Yaskawa INFORM job: X2_DOD_HARDOX_2(90,0).JBI

/JOB
//NAME X2_DOD_HARDOX_2(90,0)
//POS
///NPOS 304,304,304,21,0,0
///TOOL 0
///POSTYPE PULSE
///PULSE
C00000=3322,-122452,-100913,-73,83322,449
C00001=-124273,-75019,-76743,-2114,92937,4431
C00002=-124273,-75019,-76743,-2114,92937,4431
C00003=-142747,-87673,-78422,-11081,73870,-1911
C00004=-145871,-78515,-73342,-10252,75010,-3119
C00005=-145871,-78057,-71113,-10305,73892,-3025
C00006=-145871,-78160,-71592,-10294,74129,-3045
C00007=-146817,-82702,-73614,-10112,72935,-3281
C00008=-146817,-82536,-72956,-10129,72622,-3254
C00009=-146351,-80344,-71991,-10217,73205,-3137
C00010=-146503,-81415,-73793,-10153,73736,-3236
C00011=-173681,-53943,-60859,-2823,77659,-12885
C00012=-172671,-51589,-58765,-3102,77620,-12536
C00013=-172671,-51554,-57664,-3107,76961,-12521
C00014=-172671,-51565,-57945,-3107,77128,-12524
C00015=-174022,-54662,-59696,-2740,76567,-12973
C00016=-174022,-54640,-59313,-2741,76344,-12967
C00017=-173392,-53212,-58511,-2912,76607,-12757
C00018=-173883,-54397,-60894,-2769,77446,-12944
C00019=-147040,-82605,-78375,-9928,75852,-3597
C00020=-132076,40230,-4897,683,98086,2101
C00021=-105830,92528,44340,-4181,95198,10460
C00022=-106138,94277,47448,-496,93535,10964
C00023=-106138,93998,47888,-496,93120,10965
C00024=-106138,94075,47763,-496,93235,10965
C00025=-105307,90459,43162,-653,94213,11226
C00026=-105307,90308,43383,-653,93999,11227
C00027=-105813,92521,46192,-557,93406,11067
C00028=-105722,91355,42660,-575,94982,11088
C00029=-127942,50635,1718,3631,99633,4134
C00030=-128777,53313,5697,3773,98596,3841
C00031=-128777,52881,6272,3769,98023,3823
C00032=-128777,53071,6015,3771,98280,3831
C00033=-128282,49361,1922,3687,98870,4004
C00034=-128282,49094,2270,3685,98519,3992
C00035=-128695,51041,4408,3756,98223,3854
C00036=-128753,50417,1446,3786,99725,3882
C00037=-118729,55571,7259,-19388,105548,16023
C00038=-120440,58803,13122,-19008,103337,15802
C00039=-120440,58345,13854,-18947,102687,15906
C00040=-120440,58565,13494,-18977,103004,15855
C00041=-119879,55504,10038,-19088,103648,15942
C00042=-119879,55232,10465,-19050,103267,16004
C00043=-120241,57097,12564,-18980,102872,15943
C00044=-120239,56956,10395,-19097,104069,15748
C00045=-118897,62153,16326,-19147,103430,16312
C00046=-118943,61407,17551,-19042,102345,16473
C00047=-119386,61378,17519,-18997,102254,16335
C00048=-119201,61466,15074,-19157,103763,16154
C00049=-124650,52061,4961,-18662,103920,14273
C00050=-125121,51789,5517,-18560,103365,14201
C00051=-125121,51395,6094,-18510,102835,14285
C00052=-125121,51507,5925,-18524,102988,14260
C00053=-124425,48079,2171,-18658,103656,14391
C00054=-124425,47916,2408,-18637,103438,14425
C00055=-124770,49695,4348,-18570,103100,14361
C00056=-124479,49875,2619,-18712,104259,14276
C00057=-119059,53508,-1404,-19871,109511,15231
C00058=-119059,53508,-1404,-19871,109511,-70055
C00059=-119059,51000,874,-19526,106971,-69616
C00060=-118491,48977,220,-19515,106492,-69340
C00061=-118491,48463,842,-19443,105880,-69235
C00062=-118491,48656,606,-19469,106110,-69272
C00063=-119421,51739,3994,-19312,105438,-69476
C00064=-119421,51519,4278,-19281,105165,-69430
C00065=-119025,50120,2737,-19348,105468,-69344
C00066=-119028,51312,2337,-19442,106279,-69481
C00067=-122740,53922,5381,-20074,111685,-71721
C00068=-123083,53704,5716,-20014,111311,-71776
C00069=-123083,53271,6276,-19929,110777,-71680
C00070=-123083,53422,6076,-19958,110966,-71714
C00071=-123661,57016,10109,-19847,110240,-71793
C00072=-123661,56817,10388,-19808,109982,-71748
C00073=-123358,55142,8503,-19859,110330,-71701
C00074=-123438,56109,8263,-19951,110922,-71835
C00075=-120533,57280,6675,-20288,113056,-71184
C00076=-120494,21004,-31285,-21182,117489,-72026
C00077=-143492,-1314,-51155,-19681,113253,-79248
C00078=-143685,-8098,-52920,-19289,110944,-78908
C00079=-143685,-8785,-52225,-19179,110204,-78783
C00080=-143685,-8648,-52368,-19200,110355,-78809
C00081=-143322,-10942,-54160,-19228,110360,-78684
C00082=-143506,-8537,-54495,-19420,111686,-78976
C00083=-155354,-54452,-79937,-2145,81517,-76985
C00084=-153949,-54099,-79739,-2660,81618,-76540
C00085=-155389,-71848,-86874,-7861,69402,-77390
C00086=-156567,-71703,-86256,-7299,68995,-77772
C00087=-156567,-72078,-84796,-7350,67913,-77705
C00088=-156567,-72032,-84993,-7344,68055,-77714
C00089=-156685,-68809,-83423,-7255,68729,-77798
C00090=-157597,-72145,-85047,-6851,67942,-78069
C00091=-158988,-72221,-85084,-6184,67817,-78550
C00092=-158629,-71410,-85986,-6317,68810,-78477
C00093=-170721,-2732,-50261,-5727,95416,-85275
C00094=-178834,6538,-42419,-3288,94960,-87661
C00095=-168283,38571,-13648,-28496,116076,-28327
C00096=-172026,57706,12329,-25367,123716,-30434
C00097=-172026,57377,12858,-25209,123268,-30314
C00098=-172010,57390,12725,-25231,123353,-30330
C00099=-171834,56966,12248,-25227,123474,-30287
C00100=-172090,57867,12504,-25369,123677,-30449
C00101=-179268,34915,-13244,-27858,125223,-33968
C00102=-179209,34253,-12789,-27622,124689,-33785
C00103=-179209,33906,-12358,-27462,124294,-33669
C00104=-179209,33957,-12423,-27486,124356,-33687
C00105=-179032,33518,-12869,-27478,124454,-33639
C00106=-179236,34742,-13222,-27814,125143,-33933
C00107=-172613,57624,7301,-26510,107746,-46304
C00108=-174071,51923,5121,-34513,100734,-47012
C00109=-175632,49538,6699,-33979,98319,-46852
C00110=-175632,49118,7499,-33907,97728,-46671
C00111=-175632,49191,7354,-33918,97835,-46704
C00112=-176481,49647,7851,-33765,97460,-46913
C00113=-175632,49191,7354,-33918,97835,-46704
C00114=-175632,49191,7354,-33918,97835,-46704
C00115=-175910,45446,3305,-33927,98206,-46927
C00116=-176239,50034,6888,-33885,98213,-47051
C00117=-184945,66183,17316,-13475,101547,-47528
C00118=-185105,65696,18542,-13396,100544,-47469
C00119=-185105,65236,19213,-13363,99912,-47399
C00120=-185105,65314,19095,-13369,100021,-47411
C00121=-184391,64161,17756,-13482,100359,-47212
C00122=-185105,65314,19095,-13369,100021,-47411
C00123=-184796,67746,21947,-13388,99576,-47263
C00124=-184914,67542,19780,-13434,100755,-47432
C00125=-176930,61777,6720,-753,113886,-70793
C00126=-174340,53781,528,-827,113611,-69928
C00127=-174105,48716,-2234,-828,112710,-69842
C00128=-174105,48241,-1745,-826,112162,-69839
C00129=-174105,48415,-1929,-827,112364,-69840
C00130=-173955,52247,2291,-826,111737,-69785
C00131=-173955,52021,2539,-826,111470,-69785
C00132=-174013,49894,189,-832,111823,-69808
C00133=-173982,51573,852,-838,112278,-69801
C00134=-165923,51418,-185,4198,115847,-66019
C00135=-166041,50042,-378,4173,115265,-66082
C00136=-166041,49530,178,4148,114661,-66107
C00137=-166041,49763,-78,4158,114938,-66097
C00138=-165938,53468,4025,4136,114313,-66084
C00139=-165938,53196,4339,4123,113979,-66097
C00140=-165926,51676,2650,4131,114236,-66084
C00141=-165919,53607,2512,4172,115311,-66042
C00142=-171786,97255,45260,3933,111711,-68185
C00143=-166863,94581,46566,-26856,98023,-67956
C00144=-168209,94772,50835,-26476,95346,-67829
C00145=-168209,94538,51352,-26451,94950,-67740
C00146=-168209,94605,51200,-26457,95064,-67767
C00147=-168368,91297,46992,-26486,95816,-67996
C00148=-168209,94605,51200,-26457,95064,-67767
C00149=-175345,82615,32984,-10581,94088,-67902
C00150=-174600,81946,32154,-10748,94342,-67685
C00151=-168385,92449,47401,-26505,96117,-68071
C00152=-173055,60580,15757,-21671,81948,-66780
C00153=-173203,60112,18729,-21719,79983,-66473
C00154=-173203,59809,19432,-21753,79434,-66374
C00155=-173203,59888,19240,-21744,79581,-66401
C00156=-173218,62475,22200,-21769,79117,-66321
C00157=-173203,59888,19240,-21744,79581,-66401
C00158=-173673,59942,19303,-21577,79455,-66543
C00159=-174505,60634,20093,-21285,79126,-66772
C00160=-174264,60341,18495,-21324,79963,-66838
C00161=-167460,93103,37888,-11158,96394,-64497
C00162=-144918,43385,-1107,-8607,81861,-54431
C00163=-144528,47120,9335,-4100,76397,-53195
C00164=-144241,49530,13397,-4247,75176,-53058
C00165=-144241,49276,14314,-4260,74482,-53033
C00166=-144241,49323,14135,-4258,74615,-53038
C00167=-144298,51884,16934,-4244,74206,-53043
C00168=-144241,49323,14135,-4258,74615,-53038
C00169=-141663,39590,7124,-9995,67451,-62590
C00170=-142230,39272,6792,-9710,67425,-62790
C00171=-144241,49647,13017,-4243,75468,-53068
C00172=-146577,53893,13353,13946,80154,-68092
C00173=-146029,57800,10762,7564,81799,-68948
C00174=-146541,58593,16568,7823,78706,-69304
C00175=-146540,58247,17320,7838,78076,-69343
C00176=-146542,58320,17158,7832,78209,-69334
C00177=-146445,56045,14597,7787,78606,-69278
C00178=-146542,58320,17158,7832,78209,-69334
C00179=-145792,58980,17905,7544,78023,-69103
C00180=-146542,58637,16481,7818,78783,-69298
C00181=-144241,49530,13397,-4247,75176,-53058
C00182=-144866,51447,16596,-4012,74169,-53232
C00183=-149157,72642,30199,6740,82147,-60563
C00184=-149157,72642,30199,6740,82147,-60563
C00185=-148566,70197,27290,6539,82634,-60346
C00186=-147911,82520,33837,4028,91282,-60169
C00187=-146804,87436,38828,-1978,93451,-60942
C00188=-147097,90412,42195,-5253,94709,-61731
C00189=-147097,90412,42195,-5253,94709,-61731
C00190=-147180,72854,25212,-4939,86258,-72964
C00191=-144866,51447,16596,-4012,74169,-53232
C00192=-144558,49177,11202,-4101,76334,-53203
C00193=-151087,4830,-37169,-1451,83100,-55430
C00194=-173055,60580,15757,-21671,81948,-66780
C00195=-183199,61385,16897,-328,82159,-67424
C00196=-183796,62420,19548,802,80269,-67454
C00197=-181298,51863,9426,2718,77649,-66165
C00198=-181298,51863,9426,2718,77649,-66165
C00199=-179349,71624,27106,-690,88785,-66235
C00200=-176897,76246,31977,-4965,90770,-81100
C00201=-176127,77014,33663,-9916,89732,-81573
C00202=-178153,79021,36107,-9440,89037,-82178
C00203=-178153,79021,36107,-9440,89037,-82178
C00204=-180805,64510,21257,-4988,81800,-82147
C00205=-183796,62420,19548,802,80269,-67454
C00206=-183143,60666,16061,559,81507,-67239
C00207=-175351,25319,-26106,-2286,89371,-64908
C00208=-143492,-1314,-51155,-19681,113253,-79248
C00209=-143013,-8198,-53474,-19399,111359,-78751
C00210=-145235,-11098,-54914,-15600,110448,-78427
C00211=-151674,-13506,-56736,-14904,109260,-80393
C00212=-151674,-13506,-56736,-14904,109260,-80393
C00213=-151433,-54864,-78541,-15470,81224,-77744
C00214=-168057,-74397,-84388,7587,64049,-80279
C00215=-171701,-73671,-83029,16968,64769,-80658
C00216=-167647,-74737,-83530,14966,63764,-79277
C00217=-167647,-74737,-83530,14966,63764,-79277
C00218=-158678,-46023,-76468,3228,87512,-75789
C00219=-145235,-11098,-54914,-15600,110448,-78427
C00220=-145431,-9199,-55398,-15732,111644,-78658
C00221=-168283,39843,-14699,-28849,117224,-28651
C00222=-166811,83255,42584,-27785,123826,-28866
C00223=-167086,79755,41302,-27494,122798,-28690
C00224=-168710,71177,30960,-28573,124007,-29785
C00225=-168625,72399,31107,-28750,124512,-29903
C00226=-175338,47473,-2501,-15509,119186,-28999
C00227=-176050,44553,-4891,-13452,117513,-28654
C00228=-171753,58192,13887,-25528,123390,-30295
C00229=-176767,39085,-2637,-36678,126921,-35300
C00230=-176776,40139,-2721,-36982,127397,-35513
C00231=-182360,27126,-21127,-26354,124122,-34565
C00232=-182011,26598,-20010,-25999,123356,-34206
C00233=-178651,33093,-7598,-38814,126788,-36485
C00234=-178807,33986,-8333,-39323,127440,-36874
C00235=-171487,61662,13702,-38303,130982,-34716
C00236=-174071,51923,5121,-34513,100734,-47012
C00237=-175632,49538,6699,-33979,98319,-46852
C00238=-177380,22923,-15778,-31471,84748,-43959
C00239=-176331,36536,-2265,-31855,83983,-43359
C00240=-176331,36536,-2265,-31855,83983,-43359
C00241=-182786,57457,11953,-17173,95558,-45307
C00242=-182713,80837,37612,-15954,102904,-57013
C00243=-185235,81422,37737,-12319,106581,-57794
C00244=-186009,72888,27374,-12466,108421,-58255
C00245=-186009,72888,27374,-12466,108421,-58255
C00246=-183738,60486,13977,-18319,104700,-58054
C00247=-177380,22923,-15778,-31471,84748,-43959
C00248=-176840,23437,-17116,-31615,85870,-44074
C00249=-109818,-24177,-62499,-45723,116458,-28547
C00250=-119022,50763,-7781,-20248,111887,-70469
C00251=-117525,55267,6604,-19539,106041,-68933
C00252=-117612,60964,15080,-19605,108261,-69301
C00253=-118052,60249,14306,-19601,108267,-69458
C00254=-119038,58368,12162,-19600,108382,-69825
C00255=-124203,49673,2466,-19498,108668,-71685
C00256=-124193,51059,2241,-19612,109473,-71820
C00257=-118729,55571,7259,-19388,105548,16023
C00258=-120832,93113,53028,-13650,108421,37663
C00259=-121422,94426,55972,-13634,107554,37345
C00260=-121385,91153,51818,-13709,108413,37255
C00261=-121498,63603,18641,-13078,101888,37973
C00262=-121638,62759,17663,-13076,102030,37910
C00263=-121775,62314,17150,-13067,102096,37854
C00264=-122120,61576,16300,-13037,102186,37729
C00265=-127539,53554,7195,-12472,103203,35557
C00266=-127048,53031,4344,-12625,104724,35559
C00267=-128125,45258,-4139,3676,100479,4102
C00268=-128984,63889,14515,-6283,99846,-50505
C00269=-128973,63560,14772,-6277,99521,-50485
C00270=-128692,64260,17644,-6292,98143,-50325
C00271=-128660,63474,16732,-6301,98303,-50322
C00272=-129257,59211,12183,-5228,99293,-36352
C00273=-128256,59027,12018,-5797,101726,-20147
C00274=-130077,65460,18788,991,105658,-7094
C00275=-130302,68050,21973,4189,105347,-6636
C00276=-108723,94171,46301,2699,102932,412
C00277=-109130,78019,27714,7397,100640,1074
C00278=-108986,78619,28447,7373,100486,1112
C00279=-108874,77137,24310,7411,102248,1254
C00280=-113775,103231,45644,8140,102955,-267
C00281=-112738,67712,695,8483,112179,706
C00282=-142747,-87673,-78422,-11081,73870,-1911
C00283=-140888,-85961,-76055,-11551,73565,-1221
C00284=-139340,-68854,-68429,-12518,84827,-1847
C00285=-143950,-66538,-67268,-11865,84606,-3413
C00286=-164467,-48665,-57755,-7854,85710,-10431
C00287=-166762,-45519,-52179,-16577,77510,-11135
C00288=-166641,-47434,-54618,-16579,78031,-11163
C00289=-142747,-87673,-78422,-11081,73870,-1911
C00290=-174340,53781,528,-827,113611,-69928
C00291=-168310,39981,-12269,-15839,103749,-70486
C00292=-177645,51246,-42,-3167,110619,-71487
C00293=-177496,48519,-1117,-3157,109882,-71416
C00294=-177303,48685,-934,-3167,109864,-71352
C00295=-177224,48708,-906,-3173,109862,-71326
C00296=-176708,48575,-1049,-3204,109901,-71159
C00297=-175427,52346,3301,1034,112529,-69924
C00298=-149404,52323,3274,758,112264,-61153
C00299=-152248,56258,9669,12866,112346,-55377
C00300=-152744,58570,9760,12981,113525,-55416
C00301=-146330,6368,-43084,970,87924,-59513
C00302=-142747,-87673,-78422,-11081,73870,-1911
C00303=-124273,-75019,-76743,-2114,92937,4431
BC00000=87761,666220,1075229
BC00001=166009,666057,200053
BC00002=166009,713327,200053
BC00003=191285,720682,183381
BC00004=191285,720682,183381
BC00005=191285,720682,183381
BC00006=191285,720682,183381
BC00007=191285,720682,183381
BC00008=191285,720682,183381
BC00009=191285,720682,183381
BC00010=191285,720682,183381
BC00011=191285,720682,183381
BC00012=191285,720682,183381
BC00013=191285,720682,183381
BC00014=191285,720682,183381
BC00015=191285,720682,183381
BC00016=191285,720682,183381
BC00017=191285,720682,183381
BC00018=191285,720682,183381
BC00019=191285,720682,183381
BC00020=171167,720682,94626
BC00021=133618,734342,99
BC00022=133618,734342,99
BC00023=133618,734342,99
BC00024=133618,734342,99
BC00025=133618,734342,99
BC00026=133618,734342,99
BC00027=133618,734342,99
BC00028=133618,734342,99
BC00029=153809,734342,47664
BC00030=153809,734342,47664
BC00031=153809,734342,47664
BC00032=153809,734342,47664
BC00033=153809,734342,47664
BC00034=153809,734342,47664
BC00035=153809,734342,47664
BC00036=153809,734342,47664
BC00037=153809,734342,47664
BC00038=153809,734342,47664
BC00039=153809,734342,47664
BC00040=153809,734342,47664
BC00041=153809,734342,47664
BC00042=153809,734342,47664
BC00043=153809,734342,47664
BC00044=153809,734342,47664
BC00045=153809,734342,47664
BC00046=153809,734342,47664
BC00047=153809,734342,47664
BC00048=153809,734342,47664
BC00049=153809,734342,47664
BC00050=153809,734342,47664
BC00051=153809,734342,47664
BC00052=153809,734342,47664
BC00053=153809,734342,47664
BC00054=153809,734342,47664
BC00055=153809,734342,47664
BC00056=153809,734342,47664
BC00057=153809,734342,47664
BC00058=153809,734342,47664
BC00059=153809,734342,47664
BC00060=153809,734342,47664
BC00061=153809,734342,47664
BC00062=153809,734342,47664
BC00063=153809,734342,47664
BC00064=153809,734342,47664
BC00065=153809,734342,47664
BC00066=153809,734342,47664
BC00067=153809,734342,47664
BC00068=153809,734342,47664
BC00069=153809,734342,47664
BC00070=153809,734342,47664
BC00071=153809,734342,47664
BC00072=153809,734342,47664
BC00073=153809,734342,47664
BC00074=153809,734342,47664
BC00075=153809,734342,47664
BC00076=153809,734342,47664
BC00077=186855,734342,47664
BC00078=186855,734342,47664
BC00079=186855,734342,47664
BC00080=186855,734342,47664
BC00081=186855,734342,47664
BC00082=186855,734342,47664
BC00083=186855,734342,47664
BC00084=186855,734342,47664
BC00085=186855,734342,47664
BC00086=186855,734342,47663
BC00087=186855,734342,47663
BC00088=186855,734342,47663
BC00089=186855,734342,47663
BC00090=186855,734342,47663
BC00091=186855,734342,47663
BC00092=186855,734342,47663
BC00093=211924,758227,47663
BC00094=211924,758227,47663
BC00095=211924,758227,47663
BC00096=211924,758227,47663
BC00097=211924,758227,47663
BC00098=211924,758227,47663
BC00099=211924,758227,47663
BC00100=211924,758227,47663
BC00101=211924,758227,47663
BC00102=211924,758227,47663
BC00103=211924,758227,47663
BC00104=211924,758227,47663
BC00105=211924,758227,47663
BC00106=211924,758227,47663
BC00107=211924,758227,47663
BC00108=211923,758227,47662
BC00109=211923,758227,47662
BC00110=211923,758227,47662
BC00111=211923,758227,47662
BC00112=211923,758227,47662
BC00113=211923,758227,47662
BC00114=211923,758227,47662
BC00115=211923,758227,47662
BC00116=211923,758227,47662
BC00117=211923,758227,47662
BC00118=211923,758227,47662
BC00119=211923,758227,47662
BC00120=211923,758227,47662
BC00121=211923,758227,47662
BC00122=211923,758227,47662
BC00123=211923,758227,47662
BC00124=211923,758227,47662
BC00125=211923,758227,47662
BC00126=211923,758227,47662
BC00127=211923,758227,47662
BC00128=211923,758227,47662
BC00129=211923,758227,47662
BC00130=211923,758227,47662
BC00131=211923,758227,47662
BC00132=211923,758227,47662
BC00133=211923,758227,47662
BC00134=211923,758227,47662
BC00135=211923,758227,47662
BC00136=211923,758227,47662
BC00137=211923,758227,47662
BC00138=211923,758227,47662
BC00139=211923,758227,47662
BC00140=211923,758227,47662
BC00141=211923,758227,47662
BC00142=211923,758227,1033
BC00143=211923,758227,1033
BC00144=211923,758227,1033
BC00145=211923,758227,1033
BC00146=211923,758227,1033
BC00147=211923,758227,1033
BC00148=211923,758227,1033
BC00149=211923,758227,1033
BC00150=211923,758227,1033
BC00151=211923,758227,1033
BC00152=211923,758227,45190
BC00153=211923,758227,45190
BC00154=211923,758227,45190
BC00155=211923,758227,45190
BC00156=211923,758227,45190
BC00157=211923,758227,45190
BC00158=211923,758227,45190
BC00159=211923,758227,45190
BC00160=211923,758227,45190
BC00161=194110,758227,29
BC00162=138804,758227,92453
BC00163=138804,758227,92453
BC00164=138805,758227,92453
BC00165=138805,758227,92453
BC00166=138805,758227,92453
BC00167=138805,758227,92453
BC00168=138805,758227,92453
BC00169=138805,758227,92453
BC00170=138805,758227,92453
BC00171=138805,758227,92453
BC00172=138805,758227,92453
BC00173=142008,758227,51255
BC00174=142008,758227,51255
BC00175=142008,758227,51254
BC00176=142008,758227,51254
BC00177=142008,758227,51254
BC00178=142008,758227,51254
BC00179=142008,758227,51254
BC00180=142008,758227,51254
BC00181=138805,758227,92453
BC00182=138805,758227,92453
BC00183=153472,758227,37262
BC00184=153472,758227,37262
BC00185=153472,758227,37262
BC00186=153732,758227,23
BC00187=153732,758227,23
BC00188=153732,758227,8
BC00189=153732,758227,8
BC00190=153732,758227,12632
BC00191=138805,758227,92453
BC00192=138805,758227,92453
BC00193=138805,758227,92453
BC00194=211923,758227,45190
BC00195=211923,758227,45190
BC00196=211001,758227,45786
BC00197=210931,758227,45773
BC00198=210931,758227,45773
BC00199=210931,758227,45773
BC00200=210931,758227,45773
BC00201=210808,758227,45675
BC00202=210808,758227,45675
BC00203=210808,758227,45675
BC00204=210808,758227,45675
BC00205=211001,758227,45786
BC00206=211001,758227,45786
BC00207=211000,758226,45785
BC00208=186855,734342,47664
BC00209=186855,734342,47664
BC00210=186521,734508,47975
BC00211=186495,734527,47967
BC00212=186495,734527,47967
BC00213=186495,734527,47967
BC00214=186495,734527,47967
BC00215=186481,734537,47946
BC00216=186481,734537,47946
BC00217=186481,734537,47946
BC00218=186481,734537,47946
BC00219=186521,734508,47975
BC00220=186521,734508,47975
BC00221=211924,758227,47663
BC00222=211924,758227,47663
BC00223=211924,758227,47663
BC00224=211924,758227,47663
BC00225=211924,758227,47663
BC00226=211924,758227,47663
BC00227=211924,758227,47663
BC00228=211924,758227,47663
BC00229=211924,758227,47663
BC00230=211924,758227,47663
BC00231=211924,758227,47663
BC00232=211924,758227,47663
BC00233=211924,758227,47663
BC00234=211924,758227,47663
BC00235=211924,758227,47663
BC00236=211923,758227,47662
BC00237=211923,758227,47662
BC00238=211778,758092,47664
BC00239=211778,758092,47664
BC00240=211778,758092,47664
BC00241=211778,758092,47664
BC00242=211778,758092,47663
BC00243=211741,758059,47662
BC00244=211742,758059,47662
BC00245=211742,758059,47662
BC00246=211742,758059,47662
BC00247=211778,758092,47664
BC00248=211778,758092,47664
BC00249=138929,758092,47664
BC00250=153809,734342,47664
BC00251=153809,734342,47664
BC00252=153809,734342,47664
BC00253=153809,734342,47664
BC00254=153809,734342,47664
BC00255=153809,734342,47664
BC00256=153809,734342,47664
BC00257=153809,734342,47664
BC00258=153809,734342,47664
BC00259=153809,734342,47664
BC00260=153809,734342,47664
BC00261=153809,734342,47664
BC00262=153809,734342,47664
BC00263=153809,734342,47664
BC00264=153809,734342,47664
BC00265=153809,734342,47664
BC00266=153809,734342,47664
BC00267=153809,734342,47664
BC00268=153809,734342,47664
BC00269=153809,734342,47664
BC00270=153809,734342,47664
BC00271=153809,734342,47664
BC00272=153809,734342,47664
BC00273=153809,734342,47664
BC00274=153809,734342,47664
BC00275=153809,734342,47664
BC00276=139712,749298,1
BC00277=142771,759767,1
BC00278=142771,759767,1
BC00279=142771,759767,1
BC00280=142771,730769,1
BC00281=142771,663595,1
BC00282=191285,720682,183381
BC00283=191285,720682,183381
BC00284=191285,720682,183381
BC00285=191285,720682,183381
BC00286=191285,720682,183381
BC00287=191285,720682,183381
BC00288=191285,720682,183381
BC00289=191285,720682,183381
BC00290=211923,758227,47662
BC00291=211923,758227,47662
BC00292=211923,758227,47662
BC00293=211923,758227,47662
BC00294=211923,758227,47662
BC00295=211923,758227,47662
BC00296=211923,758227,47662
BC00297=211923,758227,47662
BC00298=171210,733220,47662
BC00299=171210,733220,47662
BC00300=171210,733220,47662
BC00301=171210,733220,47662
BC00302=191285,720682,183381
BC00303=166009,666057,200053
EC00000=798156,0
EC00001=798156,0
EC00002=798156,0
EC00003=798156,0
EC00004=798156,0
EC00005=798156,0
EC00006=798156,0
EC00007=798156,0
EC00008=798156,0
EC00009=798156,0
EC00010=798156,0
EC00011=798156,0
EC00012=798156,0
EC00013=798156,0
EC00014=798156,0
EC00015=798156,0
EC00016=798156,0
EC00017=798156,0
EC00018=798156,0
EC00019=798156,0
EC00020=798156,0
EC00021=798156,0
EC00022=798156,0
EC00023=798156,0
EC00024=798156,0
EC00025=798156,0
EC00026=798156,0
EC00027=798156,0
EC00028=798156,0
EC00029=798156,0
EC00030=798156,0
EC00031=798156,0
EC00032=798156,0
EC00033=798156,0
EC00034=798156,0
EC00035=798156,0
EC00036=798156,0
EC00037=798156,0
EC00038=798156,0
EC00039=798156,0
EC00040=798156,0
EC00041=798156,0
EC00042=798156,0
EC00043=798156,0
EC00044=798156,0
EC00045=798156,0
EC00046=798156,0
EC00047=798156,0
EC00048=798156,0
EC00049=798156,0
EC00050=798156,0
EC00051=798156,0
EC00052=798156,0
EC00053=798156,0
EC00054=798156,0
EC00055=798156,0
EC00056=798156,0
EC00057=798156,0
EC00058=798156,0
EC00059=798156,0
EC00060=798156,0
EC00061=798156,0
EC00062=798156,0
EC00063=798156,0
EC00064=798156,0
EC00065=798156,0
EC00066=798156,0
EC00067=798155,0
EC00068=798155,0
EC00069=798155,0
EC00070=798155,0
EC00071=798155,0
EC00072=798155,0
EC00073=798155,0
EC00074=798155,0
EC00075=798155,0
EC00076=798155,0
EC00077=798155,0
EC00078=798155,0
EC00079=798155,0
EC00080=798155,0
EC00081=798155,0
EC00082=798155,0
EC00083=798155,0
EC00084=798155,0
EC00085=798155,0
EC00086=798154,1
EC00087=798154,1
EC00088=798154,1
EC00089=798154,1
EC00090=798154,1
EC00091=798154,1
EC00092=798154,1
EC00093=798154,1
EC00094=798154,1
EC00095=798154,1
EC00096=798154,1
EC00097=798154,1
EC00098=798154,1
EC00099=798154,1
EC00100=798154,1
EC00101=798154,1
EC00102=798154,1
EC00103=798154,1
EC00104=798154,1
EC00105=798154,1
EC00106=798154,1
EC00107=798154,1
EC00108=798153,1
EC00109=798153,1
EC00110=798153,1
EC00111=798153,1
EC00112=798153,1
EC00113=798153,1
EC00114=798153,1
EC00115=798153,1
EC00116=798153,1
EC00117=798153,1
EC00118=798153,1
EC00119=798153,1
EC00120=798153,1
EC00121=798153,1
EC00122=798153,1
EC00123=798153,1
EC00124=798153,1
EC00125=798153,1
EC00126=798153,1
EC00127=798153,1
EC00128=798153,1
EC00129=798153,1
EC00130=798153,1
EC00131=798153,1
EC00132=798153,1
EC00133=798153,1
EC00134=798153,1
EC00135=798153,1
EC00136=798153,1
EC00137=798153,1
EC00138=798153,1
EC00139=798153,1
EC00140=798153,1
EC00141=798153,1
EC00142=798153,1
EC00143=798153,1
EC00144=798153,1
EC00145=798153,1
EC00146=798153,1
EC00147=798153,1
EC00148=798153,1
EC00149=798153,1
EC00150=798153,1
EC00151=798153,1
EC00152=798153,1
EC00153=798153,1
EC00154=798153,1
EC00155=798153,1
EC00156=798153,1
EC00157=798153,1
EC00158=798153,1
EC00159=798153,1
EC00160=798153,1
EC00161=798153,1
EC00162=798153,1
EC00163=798153,1
EC00164=798140,8
EC00165=798140,8
EC00166=798140,8
EC00167=798140,8
EC00168=798140,8
EC00169=798140,8
EC00170=798140,8
EC00171=798140,8
EC00172=798140,8
EC00173=798140,8
EC00174=798140,8
EC00175=798139,8
EC00176=798139,9
EC00177=798139,9
EC00178=798139,9
EC00179=798139,9
EC00180=798139,9
EC00181=798140,8
EC00182=798140,8
EC00183=798140,8
EC00184=798140,8
EC00185=798140,8
EC00186=798140,8
EC00187=798140,8
EC00188=798140,8
EC00189=798140,8
EC00190=798140,8
EC00191=798140,8
EC00192=798140,8
EC00193=798140,8
EC00194=798153,1
EC00195=798153,1
EC00196=798153,1
EC00197=798153,2
EC00198=798153,2
EC00199=798153,2
EC00200=798153,2
EC00201=798153,2
EC00202=798153,2
EC00203=798153,2
EC00204=798153,2
EC00205=798153,1
EC00206=798153,1
EC00207=798152,2
EC00208=798155,0
EC00209=798155,0
EC00210=798155,0
EC00211=798155,0
EC00212=798155,0
EC00213=798155,0
EC00214=798155,0
EC00215=798155,0
EC00216=798155,0
EC00217=798155,0
EC00218=798155,0
EC00219=798155,0
EC00220=798155,0
EC00221=798154,1
EC00222=798154,1
EC00223=798153,2
EC00224=798154,1
EC00225=798154,1
EC00226=798154,1
EC00227=798154,1
EC00228=798154,1
EC00229=798154,1
EC00230=798154,1
EC00231=798154,1
EC00232=798154,1
EC00233=798154,1
EC00234=798154,1
EC00235=798154,1
EC00236=798153,1
EC00237=798153,1
EC00238=798153,1
EC00239=798153,1
EC00240=798153,1
EC00241=798153,1
EC00242=798153,1
EC00243=798152,2
EC00244=798151,3
EC00245=798151,3
EC00246=798151,3
EC00247=798153,1
EC00248=798153,1
EC00249=798153,1
EC00250=798156,0
EC00251=798156,0
EC00252=798156,0
EC00253=798156,0
EC00254=798156,0
EC00255=798156,0
EC00256=798156,0
EC00257=798156,0
EC00258=798156,0
EC00259=798156,0
EC00260=798156,0
EC00261=798156,0
EC00262=798156,0
EC00263=798156,0
EC00264=798156,0
EC00265=798156,0
EC00266=798156,0
EC00267=798156,0
EC00268=798156,0
EC00269=798156,0
EC00270=798156,0
EC00271=798156,0
EC00272=798156,0
EC00273=798156,0
EC00274=798156,0
EC00275=798156,0
EC00276=798156,0
EC00277=798156,0
EC00278=798156,0
EC00279=798156,0
EC00280=798156,0
EC00281=798156,0
EC00282=798156,0
EC00283=798156,0
EC00284=798156,0
EC00285=798156,0
EC00286=798156,0
EC00287=798156,0
EC00288=798156,0
EC00289=798156,0
EC00290=798153,1
EC00291=798153,1
EC00292=798153,1
EC00293=798153,1
EC00294=798153,1
EC00295=798153,1
EC00296=798153,1
EC00297=798153,1
EC00298=798153,1
EC00299=798153,1
EC00300=798153,1
EC00301=798153,1
EC00302=798156,0
EC00303=798156,0
///POSTYPE BASE
///RECTAN
///RCONF 0,0,0,0,0,0,0,0,0,0,0,0,0,0,0,0,0,0,0,0,0,0,0,0
P00006=0.222,-3.123,-1.508,0.0000,0.0000,0.0000
P00021=-0.225,-6.128,-0.405,0.0000,0.0000,0.0000
P00022=0.222,-3.123,-1.508,0.0000,0.0000,0.0000
P00023=0.143,-0.036,0.682,0.0000,0.0000,0.0000
P00024=0.145,-0.552,1.326,0.0000,0.0000,0.0000
P00025=-2.003,0.006,0.728,0.0000,0.0000,0.0000
P00026=0.562,-0.002,-0.337,0.0000,0.0000,0.0000
P00027=-0.746,0.015,-9.096,0.0000,0.0000,0.0000
P00028=-2.237,-0.018,-7.702,0.0000,0.0000,0.0000
P00029=-2.156,-0.086,-4.681,0.0000,0.0000,0.0000
P00030=5.926,-4.294,-1.390,0.0000,0.0000,0.0000
P00031=1.853,-0.001,-1.549,0.0000,0.0000,0.0000
P00032=1.957,0.503,-7.217,0.0000,0.0000,0.0000
///RCONF 0,0,0,0,1,0,0,0,0,0,0,0,0,0,0,0,0,0,0,0,0,0,0,0
P00033=-0.123,0.612,-5.012,0.0000,0.0000,0.0000
///RCONF 0,0,0,0,0,0,0,0,0,0,0,0,0,0,0,0,0,0,0,0,0,0,0,0
P00034=-0.304,0.773,-2.693,0.0000,0.0000,0.0000
P00035=2.817,0.591,-1.622,0.0000,0.0000,0.0000
P00036=-1.108,-0.829,1.850,0.0000,0.0000,0.0000
P00037=0.023,0.937,-2.677,0.0000,0.0000,0.0000
P00038=0.158,-1.133,-1.952,0.0000,0.0000,0.0000
P00039=0.012,-3.081,-0.106,0.0000,0.0000,0.0000
P00040=-0.030,9.648,2.467,0.0000,0.0000,0.0000
//INST
///DATE 2025/03/18 10:13
///ATTR SC,RW
///GROUP1 RB1,BS1
///GROUP2 ST1
NOP
MOVJ C00000 BC00000 VJ=100.00  +MOVJ EC00000 VJ=100.00
MOVJ C00001 BC00001 VJ=100.00  +MOVJ EC00001 VJ=100.00
SFTOF3D
MOVJ C00002 BC00002 VJ=100.00  +MOVJ EC00002 VJ=100.00
MOVL C00003 BC00003 V=800.0  +MOVJ EC00003 VJ=100.00
SMOVL C00004 BC00004 V=166.7  +MOVJ EC00004
SREFP 3 C00005 BC00005  +REFP EC00005
CALL JOB:SEARCH-R1-S13D
SET P022 P006
SFTON3D P022
SMOVL C00006 BC00006 V=166.7  +MOVJ EC00006
SMOVL C00007 BC00007 V=166.7  +MOVJ EC00007
MOVL C00008 BC00008 V=166.7  +MOVJ EC00008 VJ=50.00
SREFP 3 C00009 BC00009  +REFP EC00009
CALL JOB:SEARCH-R1-S13D
SET P022 P006
SFTON3D P022
SMOVL C00010 BC00010 V=166.7  +MOVJ EC00010
SFTOF3D
MOVL C00011 BC00011 V=800.0  +MOVJ EC00011 VJ=100.00
SMOVL C00012 BC00012 V=166.7  +MOVJ EC00012
SREFP 3 C00013 BC00013  +REFP EC00013
CALL JOB:SEARCH-R1-S13D
SET P021 P006
SFTON3D P021
SMOVL C00014 BC00014 V=166.7  +MOVJ EC00014
SMOVL C00015 BC00015 V=166.7  +MOVJ EC00015
MOVL C00016 BC00016 V=166.7  +MOVJ EC00016 VJ=50.00
SREFP 3 C00017 BC00017  +REFP EC00017
CALL JOB:SEARCH-R1-S13D
SET P021 P006
SFTON3D P021
SMOVL C00018 BC00018 V=166.7  +MOVJ EC00018
MOVL C00019 BC00019 V=800.0  +MOVJ EC00019 VJ=50.00
MOVL C00020 BC00020 V=800.0  +MOVJ EC00020 VJ=50.00
MOVL C00021 BC00021 V=800.0  +MOVJ EC00021 VJ=50.00
SMOVL C00022 BC00022 V=166.7  +MOVJ EC00022
SREFP 3 C00023 BC00023  +REFP EC00023
CALL JOB:SEARCH-R1-S13D
SET P023 P006
SFTON3D P023
SMOVL C00024 BC00024 V=166.7  +MOVJ EC00024
SMOVL C00025 BC00025 V=166.7  +MOVJ EC00025
MOVL C00026 BC00026 V=166.7  +MOVJ EC00026 VJ=50.00
SREFP 3 C00027 BC00027  +REFP EC00027
CALL JOB:SEARCH-R1-S13D
SET P023 P006
SFTON3D P023
SMOVL C00028 BC00028 V=166.7  +MOVJ EC00028
SFTOF3D
MOVL C00029 BC00029 V=800.0  +MOVJ EC00029 VJ=100.00
SMOVL C00030 BC00030 V=166.7  +MOVJ EC00030
SREFP 3 C00031 BC00031  +REFP EC00031
CALL JOB:SEARCH-R1-S13D
SET P024 P006
SFTON3D P024
SMOVL C00032 BC00032 V=166.7  +MOVJ EC00032
SMOVL C00033 BC00033 V=166.7  +MOVJ EC00033
MOVL C00034 BC00034 V=166.7  +MOVJ EC00034 VJ=50.00
SREFP 3 C00035 BC00035  +REFP EC00035
CALL JOB:SEARCH-R1-S13D
SET P024 P006
SFTON3D P024
SMOVL C00036 BC00036 V=166.7  +MOVJ EC00036
SFTOF3D
MOVL C00037 BC00037 V=800.0  +MOVJ EC00037 VJ=100.00
SMOVL C00038 BC00038 V=166.7  +MOVJ EC00038
SREFP 3 C00039 BC00039  +REFP EC00039
CALL JOB:SEARCH-R1-S13D
SET P025 P006
SFTON3D P025
SMOVL C00040 BC00040 V=166.7  +MOVJ EC00040
SMOVL C00041 BC00041 V=166.7  +MOVJ EC00041
MOVL C00042 BC00042 V=166.7  +MOVJ EC00042 VJ=50.00
SREFP 3 C00043 BC00043  +REFP EC00043
CALL JOB:SEARCH-R1-S13D
SET P025 P006
SFTON3D P025
SMOVL C00044 BC00044 V=166.7  +MOVJ EC00044
SMOVL C00045 BC00045 V=166.7  +MOVJ EC00045
MOVL C00046 BC00046 V=166.7  +MOVJ EC00046 VJ=50.00
SREFP 3 C00047 BC00047  +REFP EC00047
CALL JOB:SEARCH-R1-S13D
SET P025 P006
SFTON3D P025
SMOVL C00048 BC00048 V=166.7  +MOVJ EC00048
SFTOF3D
MOVL C00049 BC00049 V=800.0  +MOVJ EC00049 VJ=100.00
SMOVL C00050 BC00050 V=166.7  +MOVJ EC00050
SREFP 3 C00051 BC00051  +REFP EC00051
CALL JOB:SEARCH-R1-S13D
SET P026 P006
SFTON3D P026
SMOVL C00052 BC00052 V=166.7  +MOVJ EC00052
SMOVL C00053 BC00053 V=166.7  +MOVJ EC00053
MOVL C00054 BC00054 V=166.7  +MOVJ EC00054 VJ=50.00
SREFP 3 C00055 BC00055  +REFP EC00055
CALL JOB:SEARCH-R1-S13D
SET P026 P006
SFTON3D P026
SMOVL C00056 BC00056 V=166.7  +MOVJ EC00056
SFTOF3D
MOVL C00057 BC00057 V=800.0  +MOVJ EC00057 VJ=50.00
MOVJ C00058 BC00058 VJ=100.00  +MOVJ EC00058 VJ=50.00
MOVL C00059 BC00059 V=800.0  +MOVJ EC00059 VJ=100.00
SMOVL C00060 BC00060 V=166.7  +MOVJ EC00060
SREFP 3 C00061 BC00061  +REFP EC00061
CALL JOB:SEARCH-R1-S13D
SET P027 P006
SFTON3D P027
SMOVL C00062 BC00062 V=166.7  +MOVJ EC00062
SMOVL C00063 BC00063 V=166.7  +MOVJ EC00063
MOVL C00064 BC00064 V=166.7  +MOVJ EC00064 VJ=50.00
SREFP 3 C00065 BC00065  +REFP EC00065
CALL JOB:SEARCH-R1-S13D
SET P027 P006
SFTON3D P027
SMOVL C00066 BC00066 V=166.7  +MOVJ EC00066
SFTOF3D
MOVL C00067 BC00067 V=800.0  +MOVJ EC00067 VJ=100.00
SMOVL C00068 BC00068 V=166.7  +MOVJ EC00068
SREFP 3 C00069 BC00069  +REFP EC00069
CALL JOB:SEARCH-R1-S13D
SET P028 P006
SFTON3D P028
SMOVL C00070 BC00070 V=166.7  +MOVJ EC00070
SMOVL C00071 BC00071 V=166.7  +MOVJ EC00071
MOVL C00072 BC00072 V=166.7  +MOVJ EC00072 VJ=50.00
SREFP 3 C00073 BC00073  +REFP EC00073
CALL JOB:SEARCH-R1-S13D
SET P028 P006
SFTON3D P028
SMOVL C00074 BC00074 V=166.7  +MOVJ EC00074
SFTOF3D
MOVL C00075 BC00075 V=800.0  +MOVJ EC00075 VJ=100.00
MOVL C00076 BC00076 V=800.0  +MOVJ EC00076 VJ=100.00
MOVL C00077 BC00077 V=800.0  +MOVJ EC00077 VJ=100.00
SMOVL C00078 BC00078 V=166.7  +MOVJ EC00078
SREFP 3 C00079 BC00079  +REFP EC00079
CALL JOB:SEARCH-R1-S13D
SET P031 P006
SFTON3D P031
SMOVL C00080 BC00080 V=166.7  +MOVJ EC00080
SREFP 3 C00081 BC00081  +REFP EC00081
CALL JOB:SEARCH-R1-S13D
SET P031 P006
SFTON3D P031
SMOVL C00082 BC00082 V=166.7  +MOVJ EC00082
SMOVL C00083 BC00083 V=166.7  +MOVJ EC00083
SREFP 3 C00084 BC00084  +REFP EC00084
CALL JOB:SEARCH-R1-S13D
SET P031 P006
SFTON3D P031
MOVL C00085 BC00085 V=800.0  +MOVJ EC00085 VJ=100.00
SMOVL C00086 BC00086 V=166.7  +MOVJ EC00086
SREFP 3 C00087 BC00087  +REFP EC00087
CALL JOB:SEARCH-R1-S13D
SET P032 P006
SFTON3D P032
SMOVL C00088 BC00088 V=166.7  +MOVJ EC00088
SREFP 3 C00089 BC00089  +REFP EC00089
CALL JOB:SEARCH-R1-S13D
SET P032 P006
SFTON3D P032
SMOVL C00090 BC00090 V=166.7  +MOVJ EC00090
SREFP 3 C00091 BC00091  +REFP EC00091
CALL JOB:SEARCH-R1-S13D
SET P032 P006
SFTON3D P032
SMOVL C00092 BC00092 V=166.7  +MOVJ EC00092
MOVL C00093 BC00093 V=800.0  +MOVJ EC00093 VJ=100.00
MOVL C00094 BC00094 V=800.0  +MOVJ EC00094 VJ=100.00
MOVJ C00095 BC00095 VJ=100.00  +MOVJ EC00095 VJ=100.00
SMOVL C00096 BC00096 V=166.7  +MOVJ EC00096
SREFP 3 C00097 BC00097  +REFP EC00097
CALL JOB:SEARCH-R1-S13D
SET P034 P006
SFTON3D P034
SMOVL C00098 BC00098 V=166.7  +MOVJ EC00098
SREFP 3 C00099 BC00099  +REFP EC00099
CALL JOB:SEARCH-R1-S13D
SET P034 P006
SFTON3D P034
SMOVL C00100 BC00100 V=166.7  +MOVJ EC00100
MOVL C00101 BC00101 V=800.0  +MOVJ EC00101 VJ=100.00
SMOVL C00102 BC00102 V=166.7  +MOVJ EC00102
SREFP 3 C00103 BC00103  +REFP EC00103
CALL JOB:SEARCH-R1-S13D
SET P033 P006
SFTON3D P033
SMOVL C00104 BC00104 V=166.7  +MOVJ EC00104
SREFP 3 C00105 BC00105  +REFP EC00105
CALL JOB:SEARCH-R1-S13D
SET P033 P006
SFTON3D P033
SMOVL C00106 BC00106 V=166.7  +MOVJ EC00106
SFTOF3D
MOVJ C00107 BC00107 VJ=100.00  +MOVJ EC00107 VJ=100.00
MOVL C00108 BC00108 V=800.0  +MOVJ EC00108 VJ=100.00
SMOVL C00109 BC00109 V=166.7  +MOVJ EC00109
SREFP 3 C00110 BC00110  +REFP EC00110
CALL JOB:SEARCH-R1-S13D
SET P035 P006
SFTON3D P035
SMOVL C00111 BC00111 V=166.7  +MOVJ EC00111
SREFP 3 C00112 BC00112  +REFP EC00112
CALL JOB:SEARCH-R1-S13D
SET P035 P006
SFTON3D P035
SMOVL C00113 BC00113 V=166.7  +MOVJ EC00113
SMOVL C00114 BC00114 V=166.7  +MOVJ EC00114
SREFP 3 C00115 BC00115  +REFP EC00115
CALL JOB:SEARCH-R1-S13D
SET P035 P006
SFTON3D P035
SMOVL C00116 BC00116 V=166.7  +MOVJ EC00116
MOVL C00117 BC00117 V=800.0  +MOVJ EC00117 VJ=100.00
SMOVL C00118 BC00118 V=166.7  +MOVJ EC00118
SREFP 3 C00119 BC00119  +REFP EC00119
CALL JOB:SEARCH-R1-S13D
SET P036 P006
SFTON3D P036
SMOVL C00120 BC00120 V=166.7  +MOVJ EC00120
SREFP 3 C00121 BC00121  +REFP EC00121
CALL JOB:SEARCH-R1-S13D
SET P036 P006
SFTON3D P036
SMOVL C00122 BC00122 V=166.7  +MOVJ EC00122
SREFP 3 C00123 BC00123  +REFP EC00123
CALL JOB:SEARCH-R1-S13D
SET P036 P006
SFTON3D P036
SMOVL C00124 BC00124 V=166.7  +MOVJ EC00124
MOVL C00125 BC00125 V=800.0  +MOVJ EC00125 VJ=100.00
MOVL C00126 BC00126 V=800.0  +MOVJ EC00126 VJ=100.00
SMOVL C00127 BC00127 V=166.7  +MOVJ EC00127
SREFP 3 C00128 BC00128  +REFP EC00128
CALL JOB:SEARCH-R1-S13D
SET P030 P006
SFTON3D P030
SMOVL C00129 BC00129 V=166.7  +MOVJ EC00129
SMOVL C00130 BC00130 V=166.7  +MOVJ EC00130
SMOVL C00131 BC00131 V=166.7  +MOVJ EC00131
SREFP 3 C00132 BC00132  +REFP EC00132
CALL JOB:SEARCH-R1-S13D
SET P030 P006
SFTON3D P030
SMOVL C00133 BC00133 V=166.7  +MOVJ EC00133
SFTOF3D
MOVL C00134 BC00134 V=800.0  +MOVJ EC00134 VJ=100.00
SMOVL C00135 BC00135 V=166.7  +MOVJ EC00135
SREFP 3 C00136 BC00136  +REFP EC00136
CALL JOB:SEARCH-R1-S13D
SET P029 P006
SFTON3D P029
SMOVL C00137 BC00137 V=166.7  +MOVJ EC00137
SMOVL C00138 BC00138 V=166.7  +MOVJ EC00138
SMOVL C00139 BC00139 V=166.7  +MOVJ EC00139
SREFP 3 C00140 BC00140  +REFP EC00140
CALL JOB:SEARCH-R1-S13D
SET P029 P006
SFTON3D P029
SMOVL C00141 BC00141 V=166.7  +MOVJ EC00141
SFTOF3D
MOVL C00142 BC00142 V=800.0  +MOVJ EC00142 VJ=100.00
MOVL C00143 BC00143 V=800.0  +MOVJ EC00143 VJ=100.00
SMOVL C00144 BC00144 V=166.7  +MOVJ EC00144
SREFP 3 C00145 BC00145  +REFP EC00145
CALL JOB:SEARCH-R1-S13D
SET P038 P006
SFTON3D P038
SMOVL C00146 BC00146 V=166.7  +MOVJ EC00146
SREFP 3 C00147 BC00147  +REFP EC00147
CALL JOB:SEARCH-R1-S13D
SET P038 P006
SFTON3D P038
SMOVL C00148 BC00148 V=166.7  +MOVJ EC00148
SMOVL C00149 BC00149 V=166.7  +MOVJ EC00149
SREFP 3 C00150 BC00150  +REFP EC00150
CALL JOB:SEARCH-R1-S13D
SET P038 P006
SFTON3D P038
SMOVL C00151 BC00151 V=166.7  +MOVJ EC00151
MOVL C00152 BC00152 V=800.0  +MOVJ EC00152 VJ=100.00
SMOVL C00153 BC00153 V=166.7  +MOVJ EC00153
SREFP 3 C00154 BC00154  +REFP EC00154
CALL JOB:SEARCH-R1-S13D
SET P037 P006
SFTON3D P037
SMOVL C00155 BC00155 V=166.7  +MOVJ EC00155
SREFP 3 C00156 BC00156  +REFP EC00156
CALL JOB:SEARCH-R1-S13D
SET P037 P006
SFTON3D P037
SMOVL C00157 BC00157 V=166.7  +MOVJ EC00157
SMOVL C00158 BC00158 V=166.7  +MOVJ EC00158
SREFP 3 C00159 BC00159  +REFP EC00159
CALL JOB:SEARCH-R1-S13D
SET P037 P006
SFTON3D P037
SMOVL C00160 BC00160 V=166.7  +MOVJ EC00160
MOVL C00161 BC00161 V=800.0  +MOVJ EC00161 VJ=100.00
MOVL C00162 BC00162 V=800.0  +MOVJ EC00162 VJ=100.00
MOVL C00163 BC00163 V=800.0  +MOVJ EC00163 VJ=100.00
SMOVL C00164 BC00164 V=166.7  +MOVJ EC00164
SREFP 3 C00165 BC00165  +REFP EC00165
CALL JOB:SEARCH-R1-S13D
SET P039 P006
SFTON3D P039
SMOVL C00166 BC00166 V=166.7  +MOVJ EC00166
SREFP 3 C00167 BC00167  +REFP EC00167
CALL JOB:SEARCH-R1-S13D
SET P039 P006
SFTON3D P039
SMOVL C00168 BC00168 V=166.7  +MOVJ EC00168
SMOVL C00169 BC00169 V=166.7  +MOVJ EC00169
SREFP 3 C00170 BC00170  +REFP EC00170
CALL JOB:SEARCH-R1-S13D
SET P039 P006
SFTON3D P039
SMOVL C00171 BC00171 V=166.7  +MOVJ EC00171
MOVL C00172 BC00172 V=333.3  +MOVJ EC00172 VJ=100.00
MOVL C00173 BC00173 V=333.3  +MOVJ EC00173 VJ=100.00
SMOVL C00174 BC00174 V=166.7  +MOVJ EC00174
SREFP 3 C00175 BC00175  +REFP EC00175
CALL JOB:SEARCH-R1-S13D
SET P040 P006
SFTON3D P040
SMOVL C00176 BC00176 V=166.7  +MOVJ EC00176
SREFP 3 C00177 BC00177  +REFP EC00177
CALL JOB:SEARCH-R1-S13D
SET P040 P006
SFTON3D P040
SMOVL C00178 BC00178 V=166.7  +MOVJ EC00178
SREFP 3 C00179 BC00179  +REFP EC00179
CALL JOB:SEARCH-R1-S13D
SET P040 P006
SFTON3D P040
SMOVL C00180 BC00180 V=166.7  +MOVJ EC00180
SFTOF3D
MOVL C00181 BC00181 V=333.3  +MOVJ EC00181 VJ=100.00
SFTON3D P039
SMOVL C00182 BC00182 V=150.0 PL=0  +MOVJ EC00182
MACRO1 MJ#(0) ARGF9
ARCON
SFTON3D P040
SMOVL C00183 BC00183 V=11.7  +MOVJ EC00183
SMOVC C00184 BC00184 V=13.3  +MOVJ EC00184
SMOVC C00185 BC00185 V=13.3  +MOVJ EC00185
SMOVC C00186 BC00186 V=13.3  +MOVJ EC00186
SFTON3D P039
SMOVL C00187 BC00187 V=11.7  +MOVJ EC00187
SMOVL C00188 BC00188 V=11.7  +MOVJ EC00188
SMOVC C00189 BC00189 V=13.3  +MOVJ EC00189
SMOVC C00190 BC00190 V=13.3  +MOVJ EC00190
SMOVC C00191 BC00191 V=16.7  +MOVJ EC00191
ARCOF
SMOVL C00192 BC00192 V=166.7  +MOVJ EC00192
SFTOF3D
MOVL C00193 BC00193 V=800.0  +MOVJ EC00193 VJ=100.00
MOVL C00194 BC00194 V=800.0  +MOVJ EC00194 VJ=100.00
MOVL C00195 BC00195 V=333.3  +MOVJ EC00195 VJ=100.00
SFTON3D P037
SMOVL C00196 BC00196 V=150.0 PL=0  +MOVJ EC00196
ARCON
SFTON3D P038
SMOVL C00197 BC00197 V=11.7  +MOVJ EC00197
SMOVC C00198 BC00198 V=13.3  +MOVJ EC00198
SMOVC C00199 BC00199 V=13.3  +MOVJ EC00199
SMOVC C00200 BC00200 V=13.3  +MOVJ EC00200
SFTON3D P037
SMOVL C00201 BC00201 V=11.7  +MOVJ EC00201
SMOVL C00202 BC00202 V=11.7  +MOVJ EC00202
SMOVC C00203 BC00203 V=13.3  +MOVJ EC00203
SMOVC C00204 BC00204 V=13.3  +MOVJ EC00204
SMOVC C00205 BC00205 V=13.3  +MOVJ EC00205
ARCOF
SMOVL C00206 BC00206 V=166.7  +MOVJ EC00206
SFTOF3D
MOVL C00207 BC00207 V=800.0  +MOVJ EC00207 VJ=100.00
MOVL C00208 BC00208 V=800.0  +MOVJ EC00208 VJ=100.00
MOVL C00209 BC00209 V=333.3  +MOVJ EC00209 VJ=100.00
SFTON3D P031
SMOVL C00210 BC00210 V=150.0 PL=0  +MOVJ EC00210
ARCON
SFTON3D P032
SMOVL C00211 BC00211 V=11.7  +MOVJ EC00211
SMOVC C00212 BC00212 V=13.3  +MOVJ EC00212
SMOVC C00213 BC00213 V=13.3  +MOVJ EC00213
SMOVC C00214 BC00214 V=13.3  +MOVJ EC00214
SFTON3D P031
SMOVL C00215 BC00215 V=11.7  +MOVJ EC00215
SMOVL C00216 BC00216 V=11.7  +MOVJ EC00216
SMOVC C00217 BC00217 V=13.3  +MOVJ EC00217
SMOVC C00218 BC00218 V=13.3  +MOVJ EC00218
SMOVC C00219 BC00219 V=13.3  +MOVJ EC00219
ARCOF
SMOVL C00220 BC00220 V=333.3  +MOVJ EC00220
SFTOF3D
MOVJ C00221 BC00221 VJ=100.00  +MOVJ EC00221 VJ=100.00
MOVL C00222 BC00222 V=333.3  +MOVJ EC00222 VJ=100.00
SFTON3D P034
SMOVL C00223 BC00223 V=150.0 PL=0  +MOVJ EC00223
ARCON
SWVON WEV#(70)
SMOVL C00224 BC00224 V=6.7  +MOVJ EC00224
ARCOF
SWVOF
SMOVL C00225 BC00225 V=166.7  +MOVJ EC00225
SMOVL C00226 BC00226 V=166.7  +MOVJ EC00226
SMOVL C00227 BC00227 V=150.0 PL=0  +MOVJ EC00227
ARCON
SWVON WEV#(70)
SMOVL C00228 BC00228 V=6.7  +MOVJ EC00228
SFTON3D P033
SMOVL C00229 BC00229 V=6.7  +MOVJ EC00229
ARCOF
SWVOF
SMOVL C00230 BC00230 V=166.7  +MOVJ EC00230
SMOVL C00231 BC00231 V=166.7  +MOVJ EC00231
SMOVL C00232 BC00232 V=150.0 PL=0  +MOVJ EC00232
ARCON
SWVON WEV#(70)
SMOVL C00233 BC00233 V=6.7  +MOVJ EC00233
ARCOF
SWVOF
SMOVL C00234 BC00234 V=166.7  +MOVJ EC00234
SFTOF3D
MOVL C00235 BC00235 V=800.0  +MOVJ EC00235 VJ=100.00
MOVL C00236 BC00236 V=800.0  +MOVJ EC00236 VJ=100.00
SMOVL C00237 BC00237 V=166.7  +MOVJ EC00237
SFTON3D P035
SMOVL C00238 BC00238 V=150.0 PL=0  +MOVJ EC00238
ARCON
SFTON3D P036
SMOVL C00239 BC00239 V=11.7  +MOVJ EC00239
SMOVC C00240 BC00240 V=13.3  +MOVJ EC00240
SMOVC C00241 BC00241 V=13.3  +MOVJ EC00241
SMOVC C00242 BC00242 V=13.3  +MOVJ EC00242
SFTON3D P035
SMOVL C00243 BC00243 V=11.7  +MOVJ EC00243
SMOVL C00244 BC00244 V=11.7  +MOVJ EC00244
SMOVC C00245 BC00245 V=13.3  +MOVJ EC00245
SMOVC C00246 BC00246 V=13.3  +MOVJ EC00246
SMOVC C00247 BC00247 V=13.3  +MOVJ EC00247
ARCOF
SMOVL C00248 BC00248 V=333.3  +MOVJ EC00248
SFTOF3D
MOVL C00249 BC00249 V=800.0  +MOVJ EC00249 VJ=100.00
MOVJ C00250 BC00250 VJ=100.00  +MOVJ EC00250 VJ=100.00
MOVJ C00251 BC00251 VJ=100.00  +MOVJ EC00251 VJ=100.00
SFTON3D P027
SMOVL C00252 BC00252 V=150.0 PL=0  +MOVJ EC00252
ARCON
SMOVL C00253 BC00253 V=10.0  +MOVJ EC00253
SMOVL C00254 BC00254 V=10.0  +MOVJ EC00254
SFTON3D P028
SMOVL C00255 BC00255 V=11.7  +MOVJ EC00255
ARCOF
SMOVL C00256 BC00256 V=333.3  +MOVJ EC00256
SFTOF3D
MOVJ C00257 BC00257 VJ=100.00  +MOVJ EC00257 VJ=100.00
SFTON3D P025
SMOVL C00258 BC00258 V=333.3  +MOVJ EC00258
SMOVL C00259 BC00259 V=150.0 PL=0  +MOVJ EC00259
ARCON
SMOVL C00260 BC00260 V=11.7  +MOVJ EC00260
SMOVL C00261 BC00261 V=11.7  +MOVJ EC00261
SMOVL C00262 BC00262 V=11.7  +MOVJ EC00262
SMOVL C00263 BC00263 V=11.7  +MOVJ EC00263
SMOVL C00264 BC00264 V=11.7  +MOVJ EC00264
SFTON3D P026
SMOVL C00265 BC00265 V=11.7  +MOVJ EC00265
ARCOF
SMOVL C00266 BC00266 V=333.3  +MOVJ EC00266
SFTOF3D
MOVL C00267 BC00267 V=800.0  +MOVJ EC00267 VJ=100.00
MOVL C00268 BC00268 V=800.0  +MOVJ EC00268 VJ=100.00
SFTON3D P024
SMOVL C00269 BC00269 V=333.3  +MOVJ EC00269
SMOVL C00270 BC00270 V=150.0 PL=0  +MOVJ EC00270
ARCON
SMOVL C00271 BC00271 V=11.7  +MOVJ EC00271
SMOVL C00272 BC00272 V=11.7  +MOVJ EC00272
SMOVL C00273 BC00273 V=11.7  +MOVJ EC00273
SMOVL C00274 BC00274 V=11.7  +MOVJ EC00274
SMOVL C00275 BC00275 V=11.7  +MOVJ EC00275
SFTON3D P023
SMOVL C00276 BC00276 V=11.7  +MOVJ EC00276
SMOVL C00277 BC00277 V=11.7  +MOVJ EC00277
SMOVL C00278 BC00278 V=11.7  +MOVJ EC00278
ARCOF
SMOVL C00279 BC00279 V=333.3  +MOVJ EC00279
SFTOF3D
MOVL C00280 BC00280 V=800.0  +MOVJ EC00280 VJ=100.00
SMOVL C00281 BC00281 V=800.0  +MOVJ EC00281
SMOVL C00282 BC00282 V=800.0  +MOVJ EC00282
SFTON3D P022
SMOVL C00283 BC00283 V=333.3  +MOVJ EC00283
SMOVL C00284 BC00284 V=150.0 PL=0  +MOVJ EC00284
ARCON
SMOVL C00285 BC00285 V=11.7  +MOVJ EC00285
SFTON3D P021
SMOVL C00286 BC00286 V=11.7  +MOVJ EC00286
SMOVL C00287 BC00287 V=11.7  +MOVJ EC00287
ARCOF
SMOVL C00288 BC00288 V=333.3  +MOVJ EC00288
SFTOF3D
MOVL C00289 BC00289 V=800.0  +MOVJ EC00289 VJ=100.00
MOVL C00290 BC00290 V=800.0  +MOVJ EC00290 VJ=100.00
MOVL C00291 BC00291 V=800.0  +MOVJ EC00291 VJ=100.00
SFTON3D P030
SMOVL C00292 BC00292 V=333.3  +MOVJ EC00292
SMOVL C00293 BC00293 V=150.0 PL=0  +MOVJ EC00293
ARCON
SMOVL C00294 BC00294 V=11.7  +MOVJ EC00294
SMOVL C00295 BC00295 V=11.7  +MOVJ EC00295
SMOVL C00296 BC00296 V=11.7  +MOVJ EC00296
SMOVL C00297 BC00297 V=11.7  +MOVJ EC00297
SFTON3D P029
SMOVL C00298 BC00298 V=11.7  +MOVJ EC00298
SMOVL C00299 BC00299 V=11.7  +MOVJ EC00299
ARCOF
SMOVL C00300 BC00300 V=333.3  +MOVJ EC00300
SFTOF3D
MOVL C00301 BC00301 V=666.7  +MOVJ EC00301 VJ=100.00
MOVL C00302 BC00302 V=1000.0  +MOVJ EC00302 VJ=100.00
MOVJ C00303 BC00303 VJ=100.00  +MOVJ EC00303 VJ=100.00
END
